(* PLC project faults, TNI-Software ControlBuild 4.00.17 *)
(* stored: creationDateTime 2005-06-20T11:53:45-01:00 *)

FUNCTION_BLOCK cmd_equipment_library.faults
  VAR_INPUT  (* CB.group=Orders CB.kind=inputVars *)
    openCmd : BOOL := false;  (* CB.mnemonicPatternPropertyName=<SY>_CMDFW_<NU> CB.libelle=Open command to the valve *)
  END_VAR
  VAR_INPUT  (* CB.group=Sensors CB.kind=inputVars *)
    openedSensorFB : BOOL := false;  (* CB.libelle=Opened sensor feedback *)
    closedSensorFB : BOOL := false;  (* CB.libelle=Closed sensor feedback *)
  END_VAR
  VAR_INPUT  (* CB.kind=inputVars *)
    acknowledgePB : BOOL := false;  (* CB.mnemonicPatternPropertyName=<SY>PBACK<NU> CB.libelle=Acknowledgement pushbutton *)
  END_VAR
  VAR_OUTPUT  (* CB.kind=outputVars *)
    generalFault : BOOL := false;  (* CB.mnemonicPatternPropertyName=grlFlt<SY><NU> CB.libelle=General fault of the valve *)
  END_VAR
  VAR CONSTANT  (* CB.kind=parameterVars *)
    presetMvt : DINT := 4;  (* CB.mnemonicPatternPropertyName=presetMvt<SY><NU> CB.libelle=in seconds *)
    presetDiscordance : DINT := 200;  (* CB.mnemonicPatternPropertyName=presetDisc<SY><NU> CB.libelle=in milliseconds *)
  END_VAR
  VAR  (* CB.group=Faults CB.kind=overControlVars *)
    discordanceFault : BOOL := false;  (* CB.mnemonicPatternPropertyName=discFlt<SY><NU> CB.libelle=Discordance between sensors *)
    openedSensorFault : BOOL := false;  (* CB.mnemonicPatternPropertyName=openedFlt<SY><NU> CB.libelle=Opened sensor fault *)
    closedSensorFault : BOOL := false;  (* CB.mnemonicPatternPropertyName=closedFlt<SY><NU> CB.libelle=Closed sensor fault *)
  END_VAR

(* LD diagram, written out as Structured Text *)
1:
IF acknowledgePB THEN discordanceFault := FALSE; END_IF;
IF acknowledgePB THEN openedSensorFault := FALSE; END_IF;
IF acknowledgePB THEN closedSensorFault := FALSE; END_IF;
IF acknowledgePB THEN generalFault := FALSE; END_IF;
2:
ton_sec_1(IN := openCmd, PT := presetMvt);
IF ton_sec_1.Q AND NOT openedSensorFB THEN openedSensorFault := TRUE; END_IF;
ton_sec_2(IN := NOT openCmd, PT := presetMvt);
IF ton_sec_2.Q AND NOT closedSensorFB THEN closedSensorFault := TRUE; END_IF;
3:
ton_ms_3(IN := openedSensorFB AND closedSensorFB, PT := presetDiscordance);
IF ton_ms_3.Q THEN discordanceFault := TRUE; END_IF;
4:
IF discordanceFault OR openedSensorFault OR closedSensorFault THEN generalFault := TRUE; END_IF;
END_FUNCTION_BLOCK
